// TwinCAT 3 PLC project ProgrammHalle
// ProgramVersion: 3.1.4023.0
// libraries:
//   Tc2_ModbusRTU, * (Beckhoff Automation GmbH)
//   Tc2_Standard, * (Beckhoff Automation GmbH)
//   Tc2_System, * (Beckhoff Automation GmbH)
//   Tc3_BA2_Common, * (Beckhoff Automation GmbH)
//   Tc3_BACnetRev14, * (Beckhoff Automation GmbH)
//   Tc3_BA_Common, * (Beckhoff Automation GmbH)
//   Tc3_IotBase, * (Beckhoff Automation GmbH)
//   Tc3_Module, * (Beckhoff Automation GmbH)
//   TcUnit, * (www.tcunit.org)
//   OSCAT,1.1.1,RWTH Aachen University - E.ON Energy Research Center
// project tree:
//   DUTs/ E_ControlMode.TcDUT (not stored), E_PumpControlMode.TcDUT (not stored)
//   GVLs/ ADS.TcGVL (not stored), GVL.TcGVL (not stored)
//   / PlcTask.TcTTO, UnitTest.TcTTO
//   POUs/Components/ FB_ExhAirModbus.TcPOU (not stored), FB_FanBACnet.TcPOU (not stored), FB_FanControl.TcPOU, FB_FanControl.TcPOU, FB_HydMixCir.TcPOU (not stored), FB_HydThrotCir.TcPOU (not stored), FB_JetNozzle1.TcPOU (not stored), FB_JetNozzle2.TcPOU (not stored), FB_PumpBACnet.TcPOU, FB_PumpBACnet1.TcPOU (not stored), FB_PumpBACnet2.TcPOU (not stored), FB_PumpWiloIF.TcPOU (not stored), FB_RoomControlUnit.TcPOU (not stored), FB_SenTempEL321x.TcPOU (not stored), FB_TempSensPt100.TcPOU (not stored), FB_TVJModbusMaster.TcPOU (not stored), FB_TVRModbusMaster.TcPOU (not stored), FB_ValveBACnet.TcPOU (not stored), FB_Valve_0_10V.TcPOU (not stored), FB_Valve_2_10V.TcPOU (not stored), FB_Valve_4_20A.TcPOU (not stored), FB_VFCModbus1.TcPOU (not stored), FB_VFCModbus2.TcPOU (not stored), FB_VVS_JN.TcPOU (not stored), FC_CoolingCurve.TcPOU (not stored), FC_Current4_20Raw_TO_Percentage.TcPOU (not stored), FC_HeatingCurve.TcPOU, FC_MeanOfArray.TcPOU (not stored), FC_Percentage_TO_Current4_20Raw.TcPOU (not stored), FC_Percentage_TO_Voltage0_10Raw.TcPOU (not stored), FC_Percentage_TO_Voltage2_10Raw.TcPOU (not stored), FC_Pt100Raw_TO_Temperature.TcPOU (not stored), FC_Voltage0_10Raw_TO_Percentage.TcPOU (not stored), FC_Voltage2_10Raw_TO_Percentage.TcPOU (not stored)
//   POUs/EnvTemperature/ FB_AmbientAir.TcPOU (not stored)
//   POUs/HeatSupplySystem/ FB_HSS.TcPOU (not stored), FB_HSSController.TcPOU (not stored)
//   POUs/Interfaces/ I_Controller.TcIO (not stored), I_HydraulicMixingControl.TcIO (not stored), I_HydraulicThrottlingControl.TcIO (not stored), I_JetNozzle.TcIO (not stored), I_Pump.TcIO (not stored), I_TemperatureSensor.TcIO (not stored), I_Valve.TcIO (not stored), I_VolumeFlowController.TcIO (not stored)
//   POUs/ MAIN.TcPOU (not stored)
//   POUs/SensorData/ FB_SenDaHydMixCir.TcPOU (not stored)
//   POUs/Test/Components_Test/ FC_HeatingCurve_Test.TcPOU
//   POUs/Test/HeatSupplySystem_Test/ FB_HSSController_Test.TcPOU (not stored)
//   POUs/Test/ PRG_TEST.TcPOU

CONFIGURATION ProgrammHalle
    RESOURCE PLC ON TwinCAT3
        TASK PlcTask(INTERVAL := T#10ms, PRIORITY := 20);
        TASK UnitTest(INTERVAL := T#10ms, PRIORITY := 1);
        PROGRAM MAIN WITH PlcTask : MAIN;
        PROGRAM PRG_TEST WITH UnitTest : PRG_TEST;
    END_RESOURCE
END_CONFIGURATION

// ---- POUs/Test/PRG_TEST.TcPOU
PROGRAM PRG_TEST
VAR
	HeatingCurve_Test : FC_HeatingCurve_Test;							 
END_VAR

TcUnit.RUN();

END_PROGRAM

// ---- POUs/Test/Components_Test/FC_HeatingCurve_Test.TcPOU
FUNCTION_BLOCK FC_HeatingCurve_Test EXTENDS TcUnit.FB_TestSuite // This block calls the different Test methods
VAR
END_VAR

TAmbNegative();
TAmbZero();
HeatingCurveZero();
HeatingCurveNegative();

METHOD HeatingCurveNegative // This method checks whether the heating curve can have a negative value
VAR
	HeatingCurveRes: Real;		//Actual value for Heating Curve
	ExpectedValue : REAL := -1;	//Expected value for Heating Curve
	fSlope: REAL := -1;				//Slope of Heating Curve
	fOffset: REAL := 35;				//Offset of Heating Curve
END_VAR
TEST('HeatingCurveNegative');
 
HeatingCurveRes := FC_HeatingCurve(fTempAmb := 36, fSlope, fOffset);
 
AssertEquals(Expected := ExpectedValue,
             Actual := HeatingCurveRes,
             Message := 'The calculation is not correct');
 
TEST_FINISHED();
END_METHOD

METHOD HeatingCurveZero // This method checks whether the heating curve can have zero as value
VAR
	HeatingCurveRes: REAL;		//Actual value for Heating Curve
	ExpectedValue : REAL := 0;  //Expected value for Heating Curve
	fSlope: REAL := -1;				//Slope of Heating Curve
	fOffset: REAL := 35;				//Offset of Heating Curve
//	fTempAmb: REAL

END_VAR
TEST('HeatingCurveZero');
 
HeatingCurveRes := FC_HeatingCurve(fTempAmb := 35, fSlope, fOffset);
 
AssertEquals(Expected := ExpectedValue,
             Actual := HeatingCurveRes,
             Message := 'The calculation is not correct');
 
TEST_FINISHED();
END_METHOD

METHOD TAmbNegative // This method checks whether negative ambient temperatures work properly
VAR
	HeatingCurveRes: REAL;		 //Actual value for Heating Curve
	ExpectedValue : REAL := 40;  //Expected value for Heating Curve
	fSlope: REAL := -1;				 //Slope of Heating Curve
	fOffset: REAL := 35;				 //Offset of Heating Curve
END_VAR
TEST('TAmbNegative');
 
HeatingCurveRes := FC_HeatingCurve(fTempAmb := -5, fSlope, fOffset);
 
AssertEquals(Expected := ExpectedValue,
             Actual := HeatingCurveRes,
             Message := 'The calculation is not correct');
 
TEST_FINISHED();
END_METHOD

METHOD TAmbZero // This method checks whether zero degrees as ambient temperature work properly
VAR
	HeatingCurveRes : REAL;		  //Actual value for Heating Curve
	ExpectedValue : REAL := 36;   //Expected value for Heating Curve
	fSlope: REAL := -1;				  //Slope of Heating Curve	
	fOffset: REAL := 35;				  //Offset of Heating Curve

END_VAR
TEST('TAmbZero');
 
HeatingCurveRes := FC_HeatingCurve(fTempAmb := 0, fSlope, fOffset);
 
AssertEquals(Expected := ExpectedValue,
             Actual := HeatingCurveRes,
             Message := 'The calculation is not correct');
 
TEST_FINISHED();
END_METHOD

END_FUNCTION_BLOCK

// ---- POUs/Components/FC_HeatingCurve.TcPOU
FUNCTION FC_HeatingCurve : REAL
VAR_INPUT
	fTempAmb 	: REAL; 		//Ambient temperature
	fSlope 		: REAL := -1; 	//Slope of heatcurve
	fOffset 	: REAL := 36;	//In °C; off set at T_amb=0°C
END_VAR
VAR
END_VAR
VAR CONSTANT 
END_VAR

FC_HeatingCurve := fSlope * fTempAmb + fOffset;

END_FUNCTION

// ---- POUs/Components/FB_FanControl.TcPOU
FUNCTION_BLOCK FB_FanControl
VAR_INPUT
	fSpeed	:	REAL;		//Fan speed setpoint 0..100%
END_VAR
VAR
	fSpeedSetRaw  AT%Q*	: INT 	:=0; 	//Raw value for terminal => send to the valve
END_VAR
VAR CONSTANT
		fFactor : REAL :=327.67;	// factor for calculating the terminal integer values (from percentage to int)
END_VAR

fSpeedSetRaw := REAL_TO_INT(fSpeed*fFactor);

END_FUNCTION_BLOCK

// ---- POUs/Components/FB_PumpBACnet.TcPOU
FUNCTION_BLOCK FB_PumpBACnet
VAR_INPUT
	fSet		:	REAL	:=	100.0;	//Percentage of maximum
	Mode		:	E_PumpControlMode;
	//Control mode: 1 - CONST_SPEED, 5 - CONST_PRESSURE, 6 - CONST_DIFFPRESS, 7 - VAR_DIFFPRESS, 12 - TEMP_VARIABLE, 13 - CONST_CONTROL
END_VAR
VAR_OUTPUT
	stInfo			:	ST_PumpInfo;  
	bInitSuccess	:	BOOL;
	bError			:	BOOL; 
END_VAR
VAR
	fSetRaw		:	REAL;
	//BACnet client
	DevPump		:	FB_BACnet_RemoteDevice;
	//BACnet values
	Setpoint	:	FB_BACnet_RemoteAnalogOutput_EX;
	ContMode	:	FB_BACnet_RemoteMultiStateOutput_EX;
	PumpOn		:	FB_BACnet_RemoteBinaryOutput_EX;
	Operating	:	FB_BACnet_RemoteBinaryInput_EX;
	EstFlow		:	FB_BACnet_RemoteAnalogInput_EX;		//Estimated volume flow
	EstPressure	:	FB_BACnet_RemoteAnalogInput_EX;		//Estimated pressure difference
	Speed		:	FB_BACnet_RemoteAnalogInput_EX;
	Power_Act  	:	FB_BACnet_RemoteAnalogInput_EX;
	PumpError	:	FB_BACnet_RemoteBinaryInput_EX;
END_VAR

//Regular operation
PumpError(RemoteDevice:=DevPump,bPresentValue=>bError);	//Read pump error status
IF DevPump.bOperational THEN
	CASE  Mode OF
	
	E_PumpControlMode.NONE:
		PumpOn(RemoteDevice:=DevPump, bNullPV:= TRUE, bEnablePV:=TRUE);		//Release BACnet Value
		ContMode(RemoteDevice:=DevPump, bNullPV:= TRUE, bEnablePV:=TRUE);	//Release BACnet Value
	
  	E_PumpControlMode.OFF:
		PumpOn(RemoteDevice:=DevPump,bPV:=FALSE,bEnablePV:=TRUE);			// switch pump off
	
	ELSE
		PumpOn(RemoteDevice:=DevPump,bPV:=TRUE,bEnablePV:=TRUE);
		ContMode(RemoteDevice:=DevPump,nPV:=INT_TO_UDINT(Mode), bNullPV:= FALSE, bEnablePV:=TRUE);	//Set to appropriate control mode
	END_CASE
END_IF
//Error handling
IF (DevPump.bError) OR (Setpoint.bError) OR (PumpOn.bError) OR (bError) THEN
		PumpOn(RemoteDevice:=DevPump, bPV:=FALSE, bEnablePV:=TRUE);	//Deactivate Pump in Error
END_IF

//Write Setpoint value
Setpoint(RemoteDevice:=DevPump,fPV:=fSet,bEnablePV:=TRUE);	//Setpoint

//current values
EstFlow(RemoteDevice:=DevPump,fPresentValue=>stInfo.fVolFlow);
Speed(RemoteDevice:=DevPump,fPresentValue=>stInfo.fSpeed);
Power_Act(RemoteDevice:=DevPump,fPresentValue=>stInfo.fPower);
EstPressure(RemoteDevice:=DevPump,fPresentValue=>stInfo.fPressDiff);
Operating(RemoteDevice:=DevPump,bPresentValue=>stInfo.bOperating);

METHOD Init : BOOL
VAR_INPUT
END_VAR
//Init Device
DevPump(
	bReset:=FALSE,
	bAutoReset:=FALSE,
	bDisableWOC:=FALSE,
	bReSubscribeCOV:=FALSE,
	bAutoResubscribe:=FALSE,
	bTriggerWOC:=FALSE,
	bReload:=FALSE
);
IF DevPump.bOperational THEN
	ContMode(RemoteDevice:=DevPump,nPV:=INT_TO_UDINT(1),bEnablePV:=TRUE);	//Set to appropriate control mode
	//PumpOn(RemoteDevice:=DevPump,fPV:=1,bEnablePV:=TRUE);	//Activate Pump
	PumpOn(RemoteDevice:=DevPump,bPV:=TRUE,bEnablePV:=TRUE);	//Activate Pump
	IF (NOT ContMode.bError) AND (NOT PumpOn.bError) THEN
		bInitSuccess	:=	TRUE;
	END_IF
END_IF
bInitSuccess := TRUE;
END_METHOD

END_FUNCTION_BLOCK

// ---- POUs/Components/FB_FanControl.TcPOU
FUNCTION_BLOCK FB_FanControl
VAR_INPUT
	fSpeed	:	REAL;		//Fan speed setpoint 0..100%
END_VAR
VAR
	fSpeedSetRaw  AT%Q*	: INT 	:=0; 	//Raw value for terminal => send to the valve
END_VAR
VAR CONSTANT
		fFactor : REAL :=327.67;	// factor for calculating the terminal integer values (from percentage to int)
END_VAR

fSpeedSetRaw := REAL_TO_INT(fSpeed*fFactor);

END_FUNCTION_BLOCK
